# EPICS autosave request: iocBoot/ioc1/dbSave/23i_KB_Vz_.req
%
% BURT Request File
%
% 23i:KB:Vz:  Horizontal KB mirror Z-positioning
%

file $(DIR)/assy.req ASSY=23i:KB:Vz
23i:KB:Vz:Base1:23
23i:KB:Vz:Base23
file $(DIR)/mtr1.req MTR1=23i:KB:mvz1
file $(DIR)/mtr1.req MTR1=23i:KB:mvz2
file $(DIR)/mtr1.req MTR1=23i:KB:mvz3
file $(DIR)/drv1.req DRV1=23i:KB:VZ1
file $(DIR)/drv1.req DRV1=23i:KB:VZ2
file $(DIR)/drv1.req DRV1=23i:KB:VZ3
file $(DIR)/axs1.req AXS1=23i:KB:VZ
file $(DIR)/axs1.req AXS1=23i:KB:VA
file $(DIR)/axs1.req AXS1=23i:KB:VR
